// TIA Portal V20 export
VAR_GLOBAL   // PLC tag table "Interface"
END_VAR
VAR_GLOBAL CONSTANT   // user constants
   "Able to Get" : Int := 1;
   Receiving : Int := 2;
   "Complete to Get" : Int := 3;
   "Able to Put" : Int := 11;
   Sending : Int := 12;
   "Complete to Put" : Int := 13;
   Auto : Int := 1;
   Manual : Int := 2;
   "No Interference" : Int := 77;
END_VAR
